FUNCTION_BLOCK FB_ParallelQueueJobContainerCreator IMPLEMENTS I_TaskCreator
VAR_INPUT
END_VAR
VAR_OUTPUT
END_VAR
VAR
END_VAR

METHOD create_future : I_Future
VAR_INPUT
	future_name	: STRING;
END_VAR
VAR
	_p_future : POINTER TO FB_ParallelQueueJobContainer;
END_VAR
_p_future := __NEW(FB_ParallelQueueJobContainer);
_p_future^.future_name := future_name;
create_future := _p_future^;
END_METHOD

METHOD destroy_future : I_Future
VAR_INPUT
	future	: I_Future;
END_VAR
VAR
	_p_future : POINTER TO FB_ParallelQueueJobContainer;
END_VAR
IF __QUERYPOINTER(future, _p_future) THEN
	__DELETE(_p_future);
	IF _p_future = 0  THEN
		destroy_future := 0;
	END_IF
END_IF
END_METHOD

END_FUNCTION_BLOCK

(* stored: Version 1.1.0.1, ProductVersion 3.1.4026.17
   POU FB_ParallelQueueJobContainerCreator: Id {9847853e-73aa-464f-b434-9aaf175e4eeb}, SpecialFunc None
   Method create_future: Id {9e874ed2-08b5-43dd-999f-e7f9cf182846}
   Method destroy_future: Id {57fce153-6118-4cd5-aa4d-c65d04a504f1} *)
